(* CODESYS project Elevator0428_RECOVERED_2025-06-24T23-27-54.project

Project tree, tasks and I/O mapping:
  Device : Elmo Platinum Maestro, Elmo Motion Control, version 1.0.0.2
    application Application
      libraries: Standard, * (System); VisuDialogs, * (System)
      task VISU_TASK (cyclic, interval 100 ms, priority 31) calls VisuElems.Visu_Prg, PLC_PRG
      task MainTask (cyclic, interval t#20ms, priority 1) calls nothing
      function block FB_Elevator [ST]: M_IsDoorOpen, M_Enter, M_IsMoving, M_LightState, M_IsAtFloor, M_DisplayNowFloor, M_DisplayNextFloor, M_Move, M_position, M_StopMoving, M_OpenDoor, M_DisElevatorState, M_DisplayDoorState, M_FloorBtnClick, M_CloseDoor
      function block FB_FreightEle [ST]: M_Apperance
      visualisation OutsideEle
      visualisation Elavator
      data type st_Elevator
      interface ITF_Counting: M_Enter
      visualisation FreightElavator
      visualisation Visualization
      interface ITF_Action: M_IsAtFloor, M_Move, M_FloorBtnClick, M_IsDoorOpen, M_position, M_StopMoving, M_IsMoving, M_OpenDoor, M_CloseDoor
      function block FB_PassenEle [ST]
      program PLC_PRG [ST]
      function block FB_Floor [ST]: M_UpBtn, M_CallEleUp, M_CallEleDown, M_Exit, M_DownBtn, M_DeterDirection
      interface ITF_Display: M_DisplayNowFloor, M_LightState, M_DisplayNextFloor, M_DisplayDoorState, M_DisElevatorState
    Maestro : Maestro, Elmo, version 1.0.0.2
  text list GlobalTextList
*)

// Device/Application/st_Elevator
TYPE st_Elevator :
STRUCT
	xKey  : ARRAY [1..5] OF BOOL;
	iFloor: BOOL;
	xEnter : BOOL;
	xExit : BOOL;
	EleState : STRING;
	ODoor :  BOOL;
	CDoor :  BOOL;
	iWay :  STRING;
	iNextFloor : STRING;
	iNowFloor : STRING;
	//ix_Start : BOOL;
END_STRUCT
END_TYPE

// Device/Application/PLC_PRG
PROGRAM PLC_PRG
VAR
	CallELeFloor:INT;
	
	
	fbElevator : ARRAY [1..uiObject] OF FB_Elevator;
	
	fbFreight : FB_FreightEle;
	fbFloors: ARRAY [0..5] OF FB_Floor;
	fbFloorPtrs : ARRAY [0..5] OF POINTER TO FB_Floor;
	
	passoutsideCount: INT:= 5;
	passengerCount : INT := 0;
	
	xKey : ARRAY[1..uiObject] OF BOOL;
	iCnt  : INT;
	bInit : BOOL := FALSE;
	
	curEle : REFERENCE TO FB_Elevator;
	curFloor : INT;
	tmp : INT;
	i: INT;
	j: INT;
	
	CalledElevator : INT;
END_VAR


VAR CONSTANT
	uiObject : INT := 4;
	FloorDistance: INT :=313;
END_VAR

//Ele position and set the positon
IF NOT bInit THEN
	bInit := TRUE;
	
	fbElevator[4] := fbFreight;
	fbElevator[4].minFloor := 0; // Don't know why freight elevator constructor not working
	fbElevator[4].maxCapacity := 5;
	
	
	fbElevator[1].iPos :=945;
	fbElevator[2].iPos :=1258;
	fbElevator[3].iPos :=1258;
	fbElevator[4].iPos :=1258;
	
	fbFloors[0].iPoss := 1571;
	fbFloors[1].iPoss := 1258;
	fbFloors[2].iPoss := 945;
	fbFloors[3].iPoss := 632;
	fbFloors[4].iPoss := 319;
	fbFloors[5].iPoss := 3;
	
	fbFloors[0].FloorNumber := 0;
	fbFloors[1].FloorNumber := 1;
	fbFloors[2].FloorNumber := 2;
	fbFloors[3].FloorNumber := 3;
	fbFloors[4].FloorNumber := 4;
	fbFloors[5].FloorNumber := 5;
	
	FOR i := 0 TO 5 BY 1 DO
		fbFloorPtrs[i]:= ADR(fbFloors[i]);   //pointer to fbFloors (used in fb_elevator)
	END_FOR
	
	FOR i := 1 TO 4 BY 1 DO
		fbElevator[i].FloorNow := fbElevator[i].M_IsAtFloor(fbFloorPtrs);
	END_FOR
	
	FOR i := 1 TO 4 BY 1 DO
		FOR j := 0 TO 5 BY 1 DO
			fbElevator[i].Floorptr[j]:=ADR(fbFloors[j]);  //pointer to fbFloors (store floor info in elevator)
		END_FOR
	END_FOR
		
		
	FOR i := 0 TO 5 BY 1 DO
		FOR j := 1 TO 4 BY 1 DO
			fbFloors[i].fbElevatorPtrs[j]:=ADR(fbElevator[j]);  //pointer to fbelevator (record ele info in Floors )
			fbFloors[i].shouldStop[j] := FALSE;
		END_FOR
	END_FOR	
END_IF

//check ele state: move/ not yet
FOR iCnt := 1 TO uiObject BY 1 DO
	curEle REF= fbElevator[iCnt];  //we are going to change the parameter in curEle some where else, so if not using ref, curEle only will be a clone object (will not update the change)
	IF curEle.M_IsMoving() THEN //moving
		tmp := curEle.M_IsAtFloor(fbFloorPtrs);
		IF  (tmp <> -1) AND tmp = curEle.TargetFloor THEN  //reach the TargetFloor (going to stop)
			fbElevator[iCnt].M_StopMoving();
		ELSE
			IF NOT fbElevator[iCnt].M_IsDoorOpen() THEN //start moving
				curEle.M_Move(fbFloors);
				fbElevator[iCnt].Light := fbElevator[iCnt].M_LightState();
				fbElevator[iCnt].iPos:= curEle.M_position(fbElevator[iCnt].iPos);
			END_IF
		END_IF
		
	ELSE // pending
		curEle.iWaitingCounter := curEle.iWaitingCounter + 1;
		IF NOT curEle.M_IsDoorOpen() OR curEle.iWaitingCounter > curEle.iMaxWaitingTime THEN
			curEle.iWaitingCounter := 0;
			curEle.M_CloseDoor();
			IF NOT (curEle.TargetFloor = -1) THEN  //has target then move
				curEle.M_Move(fbFloors);
				fbElevator[iCnt].Light := fbElevator[iCnt].M_LightState();
				fbElevator[iCnt].iPos:= curEle.M_position(fbElevator[iCnt].iPos);
			END_IF
		END_IF
	END_IF
	
//display part
	fbElevator[iCnt].M_DisplayNowFloor();
	fbElevator[iCnt].M_DisplayNextFloor();
	fbElevator[iCnt].M_DisplayDoorState();
	fbElevator[iCnt].M_DisElevatorState();

	
END_FOR

//see wether elevator has change target floor
(*FOR i := 0 TO 5 BY 1 DO
	IF fbFloors[i].M_UpBtn() OR  fbFloors[i].M_DownBtn() THEN
		CalledElevator := fbFloors[i].M_CallEleUp();
		IF NOT (CalledElevator = -1) THEN
			fbElevator[CalledElevator].M_Move(fbFloors);
		END_IF
	END_IF
END_FOR		*)

END_PROGRAM

// Device/Application/FB_Elevator
FUNCTION_BLOCK FB_Elevator IMPLEMENTS ITF_Action,ITF_Display,ITF_Counting
VAR_INPUT
	ix_Start  : BOOL;
	xKey  : ARRAY [0..5] OF BOOL;
	
	Floorptr: ARRAY[0..5] OF POINTER TO FB_Floor ;
	ODoor : BOOL;
	CDoor : BOOL;
	Enter : BOOL;
	iPos : INT;
	iPoss : INT;
	iWaitingCounter : INT;
	passoutsideCount: INT:= 5;
	passengerCount : INT := 0;
	iMove: INT:=0;
	FloorNow  : INT :=1;
	EleState : STRING;
	Light: BOOL := FALSE; 
	
	TargetFloor  :INT:= -1;
	maxFloor : INT := 5;
	minFloor : INT := 0;
	
	direction : INT := 0;
	maxCapacity : INT := 3;
	
END_VAR
VAR_OUTPUT
	
END_VAR
VAR
	//StrDir:STRING;
	DoMove: BOOL :=FALSE;
	stFloorNow  : STRING;
	stTargetFloor  :STRING :='';
	
	
	doorstate : BOOL := TRUE;  
	DoorDisplay : STRING;
	
	
		turnlight:BOOL;
	
	
	
	
    
	
	
	Speed: INT := 1;
	
	iKeyClicked : INT;
	
	currentFloor: BOOL;
	xEnter : BOOL;
	
	//ODoor :  BOOL;
	//CDoor :  BOOL;
	iWay :  STRING;
	iNextFloor : STRING;
	iNowFloor : STRING;
	
	os_Status : STRING;
	
	xDoorFullyOpen : BOOL;
	fbAutoCloseTimer : TON; 
	tDoorOpenDwellTime : TIME := T#10S;
	bAutoCloseTriggered : BOOL;
	
	bIsMoving : BOOL := FALSE;
	
	
	
	
	iMaxWaitingTime : INT := 50;

END_VAR
VAR CONSTANT
END_VAR

fbAutoCloseTimer.IN := xDoorFullyOpen;
fbAutoCloseTimer.PT := tDoorOpenDwellTime;
fbAutoCloseTimer ();

IF fbAutoCloseTimer.Q AND (DoorState = FALSE) AND NOT bAutoCloseTriggered THEN
	THIS^.M_CloseDoor(); 
	bAutoCloseTriggered := TRUE;
END_IF

maxFloor := 5;
minFloor := 1; // default For passenger Elevator

METHOD M_IsDoorOpen : BOOL
VAR_INPUT
END_VAR
M_IsDoorOpen := doorstate;
END_METHOD

METHOD M_Enter: BOOL
VAR_INPUT
	
END_VAR

VAR
	i:INT;
END_VAR
IF NOT (M_IsAtFloor(Floorptr) = -1) THEN
	IF passengerCount < maxCapacity AND NOT (Floorptr[FloorNow]^.passoutsideCount=0) AND M_IsDoorOpen() THEN
		Floorptr[FloorNow]^.passoutsideCount:=Floorptr[FloorNow]^.passoutsideCount -1 ;
		passengerCount := passengerCount +1;
		M_Enter := TRUE; 
		RETURN;
	END_IF
END_IF

	M_Enter := FALSE;
END_METHOD

METHOD M_IsMoving : BOOL
VAR_INPUT
END_VAR
M_IsMoving := bIsMoving;
END_METHOD

METHOD M_LightState : BOOL
VAR_INPUT
	
END_VAR
IF turnlight THEN
	M_LightState := TRUE;
ELSE
	M_LightState:= FALSE;
END_IF
END_METHOD

METHOD M_IsAtFloor : INT
VAR_INPUT
	fbFloorsPtr : ARRAY[0..5] OF POINTER TO FB_Floor;
END_VAR
VAR
	i : INT;
END_VAR
FOR i := 1 TO 5 BY 1 DO
	IF( ABS(iPos - fbFloorsPtr[i]^.iPoss) < 5) THEN  
		M_IsAtFloor := i;
		FloorNow := M_IsAtFloor;
		RETURN;
	END_IF
END_FOR
M_IsAtFloor := -1; // -1 represents, no floor
END_METHOD

METHOD M_DisplayNowFloor : STRING
VAR_INPUT
END_VAR
IF FloorNow > 0 AND FloorNow < 6 THEN
	M_DisplayNowFloor :=INT_TO_STRING(FloorNow);
	stFloorNow := M_DisplayNowFloor;
ELSIF FloorNow = 0 THEN
	M_DisplayNowFloor :='B1';
	stFloorNow := M_DisplayNowFloor;
ELSE 
	M_DisplayNowFloor := '';
	stFloorNow := M_DisplayNowFloor;
END_IF
END_METHOD

METHOD M_DisplayNextFloor : STRING
VAR_INPUT
END_VAR

VAR
	LastTargetFloor: INT:=6; //initial set as the max floor
	i:INT;
END_VAR
IF TargetFloor < LastTargetFloor THEN
	IF TargetFloor > 0 AND TargetFloor < 6 THEN
		M_DisplayNextFloor :=INT_TO_STRING(TargetFloor);
		stTargetFloor := M_DisplayNextFloor; //
	ELSIF TargetFloor = 0 THEN
		M_DisplayNextFloor :='B1';
		stTargetFloor := M_DisplayNextFloor;
	ELSE 
		M_DisplayNextFloor := '';
		stTargetFloor := M_DisplayNextFloor;
	END_IF
	LastTargetFloor:=TargetFloor;
END_IF
	RETURN;
END_METHOD

METHOD M_Move : INT
VAR_INPUT
	fbFloors : ARRAY[0..5] OF FB_Floor;
END_VAR
VAR
	target_pos : INT;
	i : INT;
	hasNextFloor : BOOL;
	lastdirect : INT;
END_VAR
bIsMoving := TRUE;


// Change direction
IF NOT (TargetFloor = -1) THEN
	//Light := TRUE;
	target_pos := fbFloors[TargetFloor].iPoss;   
	IF target_pos < iPos THEN
		direction := -1;  //DOWN
		turnlight:= TRUE;
	ELSIF target_pos > iPos THEN
		direction := 1; //UP
		turnlight:= TRUE;
	ELSE
		//direction := 0;
		turnlight:= FALSE;
	END_IF
	lastdirect:= direction;  // lastdirect for 
//not END_IF yet

	IF NOT ( ABS(iPos - target_pos) < 5) THEN
		iMove := iMove + THIS^.direction * speed;
	ELSE
		//reach target, reset
		turnlight := FALSE;
		FloorNow := M_IsAtFloor(FloorPtr);
		xKey[TargetFloor] := FALSE;
		TargetFloor := -1;
		
		
		// check whether there is next target floor
		hasNextFloor := FALSE;  
		FOR i := 0 TO 5 BY 1 DO
			IF xKey[i] THEN  //if there is still any being pressed, deal with the next target floor
				hasNextFloor := TRUE;
				EXIT; 
			END_IF
		END_FOR
		
	// Enter the next targer floor 
		
		IF hasNextFloor THEN
			IF direction = 1 THEN   //find up way first
				FOR i := FloorNow + 1 TO maxFloor BY 1 DO   
					IF xKey[i] THEN
						TargetFloor := i;
						EXIT;
					END_IF
				END_FOR
				IF TargetFloor = -1 THEN
					FOR i := FloorNow - 1 TO minFloor BY -1 DO
						IF xKey[i] THEN
							TargetFloor := i;
							EXIT;
						END_IF
					END_FOR
				END_IF
			ELSIF direction = -1 THEN  //or find down way 
				FOR i := FloorNow - 1 TO minFloor BY -1 DO
					IF xKey[i] THEN
						TargetFloor := i;
						EXIT;
					END_IF
				END_FOR
				IF TargetFloor = -1 THEN
					FOR i := FloorNow + 1 TO maxFloor BY 1 DO
						IF xKey[i] THEN
							TargetFloor := i;
							EXIT;
						END_IF
					END_FOR
				END_IF
			ELSE
				// should not happen
			END_IF
		END_IF
		
	//NO FloorBtn is on, looking for upBtn at any floor
		IF TargetFloor = -1 THEN 
			
				FOR i := 1 TO 5 BY 1 DO 
				 // check the floor , i represent floor dis
					IF FloorNow + i <= maxFloor THEN
						// M_UpBtn and M_DownBtn methods will change the button state
						////IF Floorptr[FloorNow + i]^.M_UpBtn() AND NOT Floorptr[FloorNow + i]^.UpEleGet THEN
						IF Floorptr[FloorNow + i]^.xUp AND NOT Floorptr[FloorNow + i]^.UpSolved THEN
							TargetFloor := FloorNow + i;
							Floorptr[FloorNow + i]^.UpSolved := TRUE;
							//Floorptr[FloorNow + i]^.xUp := TRUE;
							EXIT;
						////ELSIF  Floorptr[FloorNow + i]^.M_DownBtn() AND NOT Floorptr[FloorNow + i]^.DownEleGet THEN
						ELSIF  Floorptr[FloorNow + i]^.xDown AND NOT Floorptr[FloorNow + i]^.DownSolved THEN
							TargetFloor := FloorNow + i;
							Floorptr[FloorNow + i]^.DownSolved:= TRUE;
							//Floorptr[FloorNow + i]^.xDown := TRUE;
							EXIT;
						END_IF
					END_IF
					
					
					IF FloorNow - i >= minFloor THEN
						// M_UpBtn and M_DownBtn methods will change the button state			
						////IF Floorptr[FloorNow - i]^.M_UpBtn() AND NOT Floorptr[FloorNow - i]^.UpEleGet THEN
						IF Floorptr[FloorNow - i]^.xUp AND NOT Floorptr[FloorNow - i]^.UpSolved THEN
							TargetFloor := FloorNow - i;
							Floorptr[FloorNow - i]^.UpSolved:= TRUE;
							//Floorptr[FloorNow - i]^.xUp := TRUE;
							EXIT;
						////ELSIF  Floorptr[FloorNow - i]^.M_DownBtn() AND NOT Floorptr[FloorNow - i]^.DownEleGet THEN
						ELSIF  Floorptr[FloorNow - i]^.xDown AND NOT Floorptr[FloorNow - i]^.DownSolved THEN
							TargetFloor := FloorNow - i;
							Floorptr[FloorNow - i]^.DownSolved:= TRUE;
							//Floorptr[FloorNow - i]^.xDown := TRUE;
							EXIT;
						END_IF
					END_IF
								
				END_FOR
		END_IF
			
					
				
		//Ele just arrived, stop moving and open door
		M_StopMoving();
		M_OpenDoor();
	END_IF
END_IF //end_if is here
M_Move := iMove;
END_METHOD

METHOD M_position : INT
VAR_INPUT
	In_iPos: INT; 
END_VAR
In_iPos := In_iPos + direction * speed;
M_position := In_iPos;
END_METHOD

METHOD M_StopMoving
VAR_INPUT
END_VAR
iWaitingCounter := 0;
bIsMoving := FALSE;
Light := FALSE;
END_METHOD

METHOD M_OpenDoor : BOOL
VAR_INPUT
	
END_VAR
IF turnlight THEN
	doorstate:= FALSE;
ELSE
	doorstate:= TRUE;
END_IF

M_OpenDoor :=doorstate;
END_METHOD

METHOD M_DisElevatorState : STRING
VAR_INPUT
END_VAR

VAR_IN_OUT
END_VAR

VAR
	StrDir : STRING;
END_VAR
IF turnlight THEN
	IF THIS^.direction = -1 THEN
		StrDir := 'Going Up';
	ELSIF THIS^.direction =1 THEN
		StrDir := 'Going Down';
	END_IF
ELSE
	StrDir := 'Pending';
END_IF

THIS^.EleState := StrDir;
M_DisElevatorState := StrDir;
END_METHOD

METHOD M_DisplayDoorState : STRING
VAR_INPUT
END_VAR
IF doorstate THEN
	DoorDisplay := 'Open';
ELSE
	DoorDisplay := 'Close';
END_IF;
M_DisplayDoorState := DoorDisplay;

(*IF ODoor THEN
	DoorDisplay:='Open';
	doorstate:= TRUE;
ELSIF CDoor THEN
	DoorDisplay:='Close';
	doorstate:= FALSE;
END_IF*)
END_METHOD

METHOD M_FloorBtnClick : BOOL
VAR_INPUT
	xNumber  : INT;
END_VAR

VAR
	fbFloors : ARRAY[0..5] OF FB_Floor;
	btnPos : INT;
	targetPos : INT;
	curPos : INT;
END_VAR
fbFloors[0].iPoss := 1571;
fbFloors[1].iPoss := 1258;
fbFloors[2].iPoss := 945;
fbFloors[3].iPoss := 632;
fbFloors[4].iPoss := 319;
fbFloors[5].iPoss := 3;

IF xNumber < 0 OR xNumber > 5 THEN
	M_FloorBtnClick := FALSE;
	RETURN;
END_IF

//no targer floor and not moving yet
IF (NOT M_IsMoving()) AND TargetFloor = -1 THEN
	TargetFloor :=xNumber;
	xKey[xNumber]:=TRUE;
	bIsMoving := TRUE;

//already have TargetFloor
ELSIF NOT (TargetFloor = -1) THEN
	btnPos := fbFloors[xNumber].iPoss;
	targetPos := fBFloors[TargetFloor].iPoss;
	curPos := iPos;
	IF NOT xKey[xNumber] THEN
		xKey[xNumber] := TRUE;
		IF TargetFloor = xNumber THEN 
			// do nothing
		ELSIF curPos <= btnPos AND btnPos <= targetPos THEN  //ex: now at 2nd btnPos= 4, targetPos= 5
			TargetFloor := xNumber;  // TargetFloor update to btnPos= 4
		ELSIF curPos >= btnPos AND btnPos >= targetPos THEN  // same as above but downstairs
			TargetFloor := xNumber;
		END_IF
	ELSE 
		// try to cancel btn, not supported now
	END_IF
END_IF
END_METHOD

METHOD M_CloseDoor : BOOL
VAR_INPUT
END_VAR
doorstate := FALSE;
M_CloseDoor := doorstate;
END_METHOD

END_FUNCTION_BLOCK

// Device/Application/ITF_Action
INTERFACE ITF_Action

METHOD M_IsAtFloor : INT
VAR_INPUT
	fbFloorsPtr : ARRAY[0..5] OF POINTER TO FB_Floor;
END_VAR
END_METHOD

METHOD M_Move : INT
VAR_INPUT
	fbFloors : ARRAY[0..5] OF FB_Floor;
END_VAR
END_METHOD

METHOD M_FloorBtnClick : BOOL
VAR_INPUT
	xNumber  : INT;
END_VAR
END_METHOD

METHOD M_IsDoorOpen : BOOL
VAR_INPUT
END_VAR
END_METHOD

METHOD M_position : INT
VAR_INPUT
	In_iPos: INT; 
END_VAR
END_METHOD

METHOD M_StopMoving
VAR_INPUT
END_VAR
END_METHOD

METHOD M_IsMoving : BOOL
VAR_INPUT
END_VAR
END_METHOD

METHOD M_OpenDoor : BOOL
VAR_INPUT
END_VAR
END_METHOD

METHOD M_CloseDoor : BOOL
VAR_INPUT
END_VAR
END_METHOD

END_INTERFACE

// Device/Application/FB_Floor
FUNCTION_BLOCK FB_Floor 
VAR_INPUT
	
	FloorNumber : INT; // This indicates which floor current FB_Floor object is.

	iPoss : INT;
	passOutsideCount : INT:=5;
	
	fbElevatorPtrs : ARRAY[1..4] OF POINTER TO FB_Elevator;
	
	shouldStop : ARRAY[1..4] OF BOOL;
	
	UpEleGet : BOOL:= FALSE;
	DownEleGet : BOOL:= FALSE;
	
	UpSolved : BOOL := FALSE;
	DownSolved : BOOL := FALSE;
	
	xUp : BOOL;
	xDown : BOOL;
	
END_VAR
VAR
	
	
	
	
	xExit : BOOL;
	
	EleState : STRING;
		
END_VAR

METHOD M_UpBtn : BOOL
VAR_INPUT
END_VAR
VAR
	i:INT;
	PendingElevator: ARRAY [1..4] OF INT;
	FloorDis: ARRAY [1..4] OF INT;
	
	shortest:INT;
	EleWantedNumber : INT := -1;
END_VAR
IF xUp = TRUE OR (NOT xUp AND UpSolved) THEN
	RETURN;
END_IF

UpSolved := FALSE;
xUp:= TRUE;
//UpEleGet:= FALSE;

FOR i := 1 TO 4 BY 1 DO
// elevator moving or not
	IF  NOT fbElevatorPtrs[i]^.turnlight THEN
		PendingElevator[i]:= 1; //pending ELe
	ELSE
		PendingElevator[i]:= 0; //moving ELe
	END_IF
END_FOR

shortest := 20000;
EleWantedNumber := -1; //no elevator is assigned to come
FOR i := 1 TO 4 BY 1 DO
//Pending ELe, then pick a nearer one
	IF PendingElevator[i] = 1 THEN
		FloorDis[i]:=ABS(fbElevatorPtrs[i]^.iPos - iPoss);
		
		IF FloorDis[i] < shortest THEN
			shortest := FloorDis[i];
			EleWantedNumber := i;
			UpSolved := TRUE;
			xUp := FALSE;
		END_IF
	
	END_IF
END_FOR

IF EleWantedNumber = -1 THEN
	FOR i := 1 TO 4 BY 1 DO
		//moving ELe, comfirm Ele is two floor away
		IF PendingElevator[i] = 0 AND fbElevatorPtrs[i]^.direction =1 THEN
			IF fbElevatorPtrs[i]^.TargetFloor >= FloorNumber THEN		
				IF ABS(fbElevatorPtrs[i]^.iPos - iPoss >= 626) THEN
					EleWantedNumber:= i;  // no.i elevator needs to come
					UpSolved := TRUE;
					xUp := FALSE;
					EXIT;
				END_IF
			END_IF
		END_IF
	END_FOR
END_IF

IF (EleWantedNumber <>-1) THEN
	fbElevatorPtrs[EleWantedNumber]^.TargetFloor := FloorNumber;
END_IF

//IF (fbElevatorPtrs[EleWantedNumber]^.TargetFloor = FloorNumber) AND (fbElevatorPtrs[EleWantedNumber]^.M_IsDoorOpen) THEN
    //bUpRequested := FALSE;
//END_IF
//M_UpBtn:=xUp;
END_METHOD

METHOD M_CallEleUp :INT
VAR_INPUT
END_VAR
VAR
	i:INT;
	PendingElevator: ARRAY [1..4] OF INT;
	FloorDis: ARRAY [1..4] OF INT;
	
	shortest:INT;
	EleWantedNumber : INT := -1;
	
END_VAR
FOR i := 1 TO 4 BY 1 DO
// elevator moving or not
	IF  fbElevatorPtrs[i]^.turnlight THEN
		PendingElevator[i]:= 1; //pending ELe
	ELSE
		PendingElevator[i]:= 0; //moving ELe
	END_IF
END_FOR

shortest := 2000;
EleWantedNumber := -1; //no elevator is assigned to come
FOR i := 1 TO 4 BY 1 DO
//Pending ELe, then pick a nearer one
	IF PendingElevator[i] = 1 THEN
		FloorDis[i]:=ABS(fbElevatorPtrs[i]^.iPos - iPoss);
		
		IF FloorDis[i] < shortest THEN
			shortest := FloorDis[i];
			EleWantedNumber := i;
		END_IF
	
	END_IF
END_FOR

IF EleWantedNumber = -1 THEN
	FOR i := 1 TO 4 BY 1 DO
		//moving ELe, comfirm Ele is two floor away
		IF PendingElevator[i] = 0 AND fbElevatorPtrs[i]^.direction =1 THEN
			IF ABS(fbElevatorPtrs[i]^.iPos - iPoss >= 621) THEN
				EleWantedNumber:= i;  // no.i elevator needs to come
				EXIT;
			END_IF
		END_IF
	END_FOR
END_IF

M_CallEleUp:= EleWantedNumber;

//when reaching targetfloor, Btn light went out
END_METHOD

METHOD M_CallEleDown : INT
VAR_INPUT
END_VAR
VAR
	i:INT;
	PendingElevator: ARRAY [1..4] OF INT;
	FloorDis: ARRAY [1..4] OF INT;
	
	shortest:INT;
	EleWantedNumber : INT := -1;
	
END_VAR
FOR i := 1 TO 4 BY 1 DO
// elevator moving or not
	IF  fbElevatorPtrs[i]^.turnlight THEN
		PendingElevator[i]:= 1; //pending ELe
	ELSE
		PendingElevator[i]:= 0; //moving ELe
	END_IF
END_FOR

shortest := 2000;
EleWantedNumber := -1; //no elevator is assigned to come
FOR i := 1 TO 4 BY 1 DO
//Pending ELe, then pick a nearer one
	IF PendingElevator[i] = 1 THEN
		FloorDis[i]:=ABS(fbElevatorPtrs[i]^.iPos - iPoss);
		
		IF FloorDis[i] < shortest THEN
			shortest := FloorDis[i];
			EleWantedNumber := i;
			DownSolved:=TRUE;
		END_IF
	
	END_IF
END_FOR

IF EleWantedNumber = -1 THEN
	FOR i := 1 TO 4 BY 1 DO
		//moving ELe, comfirm Ele is two floor away
		IF PendingElevator[i] = 0 AND fbElevatorPtrs[i]^.direction =-1 THEN
			IF ABS(fbElevatorPtrs[i]^.iPos - iPoss >= 626) THEN
				EleWantedNumber:= i;  // no.i elevator needs to come
				DownSolved:=TRUE;
			EXIT;
			END_IF
		END_IF
	END_FOR
END_IF

M_CallEleDown:= EleWantedNumber;

//when reaching targetfloor, Btn light went out
END_METHOD

METHOD M_Exit : BOOL
VAR_INPUT
	
END_VAR
VAR
	i: INT;
END_VAR
FOR i := 1 TO 4 BY 1 DO   
	IF ( ABS(iPoss - fbElevatorPtrs[i]^.iPos) < 5) AND fbElevatorPtrs[i]^.M_IsDoorOpen() THEN
		IF fbElevatorPtrs[i]^.passengerCount > 0 AND fbElevatorPtrs[i]^.passengerCount <8 THEN
			fbElevatorPtrs[i]^.passengerCount:= fbElevatorPtrs[i]^.passengerCount-1;
			passoutsideCount:=passoutsideCount +1;
		END_IF
	END_IF
END_FOR	
(*IF passoutsideCount > 0 THEN
		FloorRef0.passoutsideCount:=FloorRef0.passoutsideCount-1;
		passengerCount := passengerCount +1;
		M_Enter := TRUE; 
	   END_IF

CASE FloorNow OF
	0: 
	
	1: IF passengerCount < maxCapacity AND NOT (FloorRef1.passoutsideCount=0) THEN
		FloorRef1.passoutsideCount:=FloorRef1.passoutsideCount-1;
		passengerCount := passengerCount +1;
		M_Enter := TRUE; 
		RETURN;
	   END_IF
	   
	2: IF passengerCount < maxCapacity AND NOT (FloorRef2.passoutsideCount=0) THEN
		FloorRef2.passoutsideCount:=FloorRef2.passoutsideCount-1;
		passengerCount := passengerCount +1;
		M_Enter := TRUE; 
		RETURN;
	   END_IF
	 
	3: IF passengerCount < maxCapacity AND NOT (FloorRef3.passoutsideCount=0) THEN
		FloorRef3.passoutsideCount:=FloorRef3.passoutsideCount-1;
		passengerCount := passengerCount +1;
		M_Enter := TRUE; 
		RETURN;
	   END_IF
	
	4: IF passengerCount < maxCapacity AND NOT (FloorRef4.passoutsideCount=0) THEN
		FloorRef4.passoutsideCount:=FloorRef4.passoutsideCount-1;
		passengerCount := passengerCount +1;
		M_Enter := TRUE; 
		RETURN;
	   END_IF
	5: IF passengerCount < maxCapacity AND NOT (FloorRef5.passoutsideCount=0) THEN
		FloorRef5.passoutsideCount:=FloorRef5.passoutsideCount-1;
		passengerCount := passengerCount +1;
		M_Enter := TRUE; 
		RETURN;
	   END_IF
	END_CASE

	M_Enter := FALSE; *)
END_METHOD

METHOD M_DownBtn : BOOL
VAR_INPUT
END_VAR
VAR
	i:INT;
	PendingElevator: ARRAY [1..4] OF INT;
	FloorDis: ARRAY [1..4] OF INT;
	
	shortest:INT;
	EleWantedNumber : INT := -1;
	
END_VAR
IF xDown = TRUE OR (NOT xDown AND DownSolved) THEN
	RETURN;
END_IF

xDown:= TRUE;
DownSolved:=FALSE;

FOR i := 1 TO 4 BY 1 DO
// elevator moving or not
	IF NOT fbElevatorPtrs[i]^.turnlight THEN
		PendingElevator[i]:= 1; //pending ELe
	ELSE
		PendingElevator[i]:= 0; //moving ELe
	END_IF
END_FOR

shortest := 20000;
EleWantedNumber := -1; //no elevator is assigned to come
FOR i := 1 TO 4 BY 1 DO
//Pending ELe, then pick a nearer one
	IF PendingElevator[i] = 1 THEN
		FloorDis[i]:=ABS(fbElevatorPtrs[i]^.iPos - iPoss);
		
		IF FloorDis[i] < shortest THEN
			shortest := FloorDis[i];
			EleWantedNumber := i;
			DownSolved := TRUE;
			xDown:= FALSE;
		END_IF
	
	END_IF
END_FOR

IF EleWantedNumber = -1 THEN
	FOR i := 1 TO 4 BY 1 DO
		//moving ELe, comfirm Ele is two floor away
		IF PendingElevator[i] = 0 AND fbElevatorPtrs[i]^.direction =-1 THEN
			IF fbElevatorPtrs[i]^.TargetFloor <= FloorNumber THEN
				IF fbElevatorPtrs[i]^.iPos - iPoss >= 626 THEN
					EleWantedNumber:= i;  // no.i elevator needs to come
					DownSolved := TRUE;
					xDown:= FALSE;
					EXIT;
				END_IF
			END_IF
		END_IF
	END_FOR
END_IF

IF NOT (EleWantedNumber= -1 )THEN
	fbElevatorPtrs[EleWantedNumber]^.TargetFloor := FloorNumber;
END_IF


//M_CallEleDown:= EleWantedNumber;

//when reaching targetfloor, Btn light went out

	
//M_DownBtn:=xDown;
END_METHOD

METHOD M_DeterDirection
VAR_INPUT
END_VAR
(*IF xUp  THEN
        direction := 1;
		Light := TRUE;
		
ELSIF xDown THEN
        direction := -1;
		Light := TRUE;
ELSE
        direction := 0;
		Light := FALSE;
END_IF;   *)
END_METHOD

END_FUNCTION_BLOCK

// Device/Application/ITF_Display
INTERFACE ITF_Display

METHOD M_DisplayNowFloor : STRING
VAR_INPUT
END_VAR
END_METHOD

METHOD M_LightState : BOOL
VAR_INPUT
	
END_VAR
END_METHOD

METHOD M_DisplayNextFloor : STRING
VAR_INPUT
END_VAR
END_METHOD

METHOD M_DisplayDoorState : STRING
VAR_INPUT
END_VAR
END_METHOD

METHOD M_DisElevatorState : STRING
VAR_INPUT
END_VAR

VAR_IN_OUT
END_VAR
END_METHOD

END_INTERFACE

// Device/Application/ITF_Counting
INTERFACE ITF_Counting

METHOD M_Enter : BOOL
VAR_INPUT
END_VAR
END_METHOD

END_INTERFACE

// Device/Application/FB_FreightEle
FUNCTION_BLOCK FB_FreightEle EXTENDS FB_Elevator
VAR_INPUT
	
END_VAR
VAR_OUTPUT
END_VAR
VAR
END_VAR

//SUPER^();
maxFloor := 5;
minFloor := 0;
maxCapacity := 5;

METHOD M_Apperance
VAR_INPUT
END_VAR
END_METHOD

END_FUNCTION_BLOCK

// Device/Application/FB_PassenEle
FUNCTION_BLOCK FB_PassenEle EXTENDS FB_Elevator 
VAR_INPUT
END_VAR
VAR_OUTPUT
END_VAR
VAR
	
END_VAR

SUPER^();
maxFloor := 5;
minFloor := 1; // default For passenger Elevator

END_FUNCTION_BLOCK

// Device/Application/OutsideEle
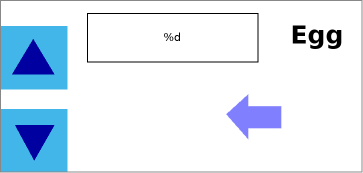
VISUALIZATION OutsideEle  // 363x173
VAR_IN_OUT
	fbFloorsVisu  : fb_Floor;
END_VAR
    RoundedRectangle (1,26 66x63)
        tap fbFloorsVisu.xUp
        OnMouseClick: execute { fbFloorsVisu.M_UpBtn(); }
    Polygon (33,39) (12,74) (54,74)
    RoundedRectangle (1,109 66x63)
        tap fbFloorsVisu.xDown
        OnMouseClick: execute { fbFloorsVisu.M_DownBtn(); }
    Polygon (15,125) (34,160) (54,125)
    Rectangle (87,13 171x49), "%d", text variable: fbFloorsVisu.passoutsideCount
    Label (292,13 50x43), "Egg"
    Polygon (226,114) (248,94) (248,106) (281,106) (281,128) (248,128) (248,139), text variable: fbFloorsVisu.xExit
        tap fbFloorsVisu.xExit
        OnMouseClick: execute { fbFloorsVisu.M_Exit(); }
END_VISUALIZATION

// Device/Application/Elavator
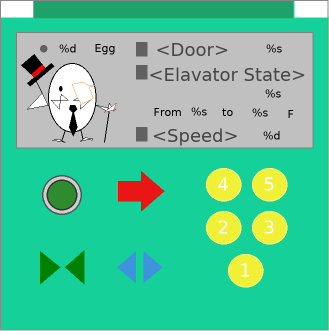
VISUALIZATION Elavator  // 329x331
VAR_IN_OUT
	fbElevatorVisu  : fb_Elevator;
END_VAR
    Polyline (46,537) (47,538)
    RoundedRectangle (0,17 329x313)
    RoundedRectangle (16,32 297x116)
    Ellipse (252,168 35x33), "5"
        tap fbElevatorVisu.xKey[5]
        OnMouseClick: execute { fbElevatorVisu.M_FloorBtnClick(5); }
    Ellipse (252,211 35x33), "3"
        tap fbElevatorVisu.xKey[3]
        OnMouseClick: execute { fbElevatorVisu.M_FloorBtnClick(3); }
    Ellipse (206,168 35x33), "4"
        tap fbElevatorVisu.xKey[4]
        OnMouseClick: execute { fbElevatorVisu.M_FloorBtnClick(4); }
    Ellipse (206,211 35x33), "2"
        tap fbElevatorVisu.xKey[2]
        OnMouseClick: execute { fbElevatorVisu.M_FloorBtnClick(2); }
    Ellipse (228,254 35x33), "1"
        tap fbElevatorVisu.xKey[1]
        OnMouseClick: execute { fbElevatorVisu.M_FloorBtnClick(1); }
    Lamp1 (39,170 46x50), variable: fbElevatorVisu.Light, style: Lamp-Lamp1-Green
    Polygon (141,171) (164,191) (141,211) (141,201) (118,201) (118,181) (141,181)
        tap fbElevatorVisu.xEnter
        OnMouseClick: execute { fbElevatorVisu.M_Enter(); }
    Rectangle (37,39 62x20), "%d", text variable: fbElevatorVisu.passengerCount
    Rectangle (136,42 11x14)
    Label (108,37 169x26), "<Door>"
    Rectangle (237,40 74x18), "%s", text variable: fbElevatorVisu.DoorDisplay
    Rectangle (223,104 74x18), "%s", text variable: fbElevatorVisu.stTargetFloor
    Rectangle (136,65 11x14)
    Label (143,62 169x26), "<Elavator State>"
    Rectangle (236,85 74x18), "%s", text variable: fbElevatorVisu.EleState
    Label (277,106 28x17), "F"
    Label (85,30 40x37), "Egg"
    Ellipse (40,45 7x7)
    Rectangle (33,0 261x19)
    Group (21,54 95x88)
        Ellipse (27,9 48x69)
        Line (41,86) (44,77)
        Line (62,85) (60,76)
        Ellipse (38,32 3x5)
        Ellipse (56,32 3x5)
        Polygon (75,51) (86,57) (88,49) (92,55)
        Polygon (69,46) (59,55) (61,42) (52,46)
        Polygon (30,46) (38,55) (40,40) (47,46)
        Polygon (15,27) (21,39) (6,55) (27,51)
        Polygon (59,87) (65,83) (71,86) (71,84)
        Line (88,55) (83,88)
        Polygon (83,58) (95,49) (92,57) (95,55)
        Polygon (31,86) (39,85) (39,86) (44,88)
        Polygon (9,32) (33,12) (30,9) (24,14) (13,0) (0,11) (13,23) (6,29)
        Polygon (13,24) (24,14) (21,10) (10,20) (13,23)
        Polygon (68,33) (72,44) (60,50) (55,41) (51,30) (62,28) (67,31) (75,31)
        Group (48,51 4x23)
            Polygon (1,0) (6,0) (8,4) (4,8) (0,4)
            Polygon (4,5) (8,22) (4,31) (0,22)
    Rectangle (162,103 74x18), "%s", text variable: fbElevatorVisu.stFloorNow
        OnMouseClick: write the text variable via Default
    Label (214,104 27x17), "to"
    Label (153,104 29x17), "From"
    Rectangle (136,127 11x14)
    Label (111,123 169x26), "<Speed>"
    Rectangle (235,127 74x18), "%d", text variable: fbElevatorVisu.Speed
        OnMouseClick: write the text variable via Default
    Polygon (137,250) (142,250) (162,267) (142,284) (137,284) (137,284) (117,267)
        tap fbElevatorVisu.ODoor
        OnMouseClick: execute { fbElevatorVisu.M_OpenDoor(); }
    Rectangle (136,240 7x50)
    Polygon (84,250) (84,284) (65,267) (60,267) (40,284) (40,251) (60,267) (65,267)
        tap fbElevatorVisu.CDoor
        OnMouseClick: execute { fbElevatorVisu.M_CloseDoor(); }
    Rectangle (61,241 3x50)
END_VISUALIZATION

// Device/Application/FreightElavator
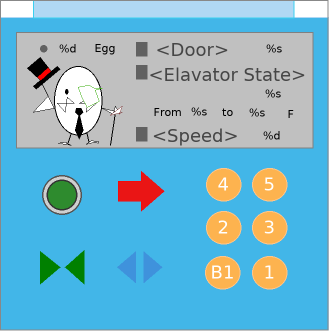
VISUALIZATION FreightElavator  // 329x331
VAR_IN_OUT
	fbFreightVisu  : FB_Elevator;
END_VAR
    Polyline (46,537) (47,538)
    RoundedRectangle (0,17 329x313)
    RoundedRectangle (16,32 297x116)
    Ellipse (252,168 35x33), "5"
        tap fbFreightVisu.xKey[5]
        OnMouseClick: execute { fbFreightVisu.M_FloorBtnClick(5); }
    Ellipse (252,211 35x33), "3"
        tap fbFreightVisu.xKey[3]
        OnMouseClick: execute { fbFreightVisu.M_FloorBtnClick(3); }
    Ellipse (206,168 35x33), "4"
        tap fbFreightVisu.xKey[4]
        OnMouseClick: execute { fbFreightVisu.M_FloorBtnClick(4); }
    Ellipse (206,211 35x33), "2"
        tap fbFreightVisu.xKey[2]
        OnMouseClick: execute { fbFreightVisu.M_FloorBtnClick(2); }
    Ellipse (252,256 35x33), "1"
        tap fbFreightVisu.xKey[1]
        OnMouseClick: execute { fbFreightVisu.M_FloorBtnClick(1); }
    Lamp1 (39,170 46x50), variable: fbFreightVisu.Light, style: Lamp-Lamp1-Green
    Polygon (141,171) (164,191) (141,211) (141,201) (118,201) (118,181) (141,181)
        tap fbFreightVisu.xEnter
        OnMouseClick: execute { fbFreightVisu.M_Enter(); }
    Rectangle (37,39 62x20), "%d", text variable: fbFreightVisu.passengerCount
    Rectangle (136,42 11x14)
    Label (108,37 169x26), "<Door>"
    Rectangle (237,40 74x18), "%s", text variable: fbFreightVisu.DoorDisplay
    Rectangle (220,104 74x18), "%s", text variable: fbFreightVisu.stTargetFloor
    Rectangle (136,65 11x14)
    Label (143,62 169x26), "<Elavator State>"
    Rectangle (236,85 74x18), "%s", text variable: fbFreightVisu.EleState
    Label (277,106 28x17), "F"
    Label (85,30 40x37), "Egg"
    Ellipse (40,45 7x7)
    Rectangle (33,-1 261x19)
    Group (27,57 95x88)
        Ellipse (27,9 48x69)
        Line (41,86) (44,77)
        Line (62,85) (60,76)
        Ellipse (38,32 3x5)
        Ellipse (56,32 3x5)
        Polygon (75,51) (86,57) (88,49) (92,55)
        Polygon (69,46) (59,55) (61,42) (52,46)
        Polygon (30,46) (38,55) (40,40) (47,46)
        Polygon (15,27) (21,39) (6,55) (27,51)
        Polygon (59,87) (65,83) (71,86) (71,84)
        Line (88,55) (83,88)
        Polygon (83,58) (95,49) (92,57) (95,55)
        Polygon (31,86) (39,85) (39,86) (44,88)
        Polygon (9,32) (33,12) (30,9) (24,14) (13,0) (0,11) (13,23) (6,29)
        Polygon (13,24) (24,14) (21,10) (10,20) (13,23)
        Polygon (68,33) (72,44) (60,50) (55,41) (51,30) (62,28) (67,31) (75,31)
        Group (48,51 4x23)
            Polygon (1,0) (6,0) (8,4) (4,8) (0,4)
            Polygon (4,5) (8,22) (4,31) (0,22)
    Rectangle (162,103 74x18), "%s", text variable: fbFreightVisu.stFloorNow
        OnMouseClick: write the text variable via Default
    Label (214,104 27x17), "to"
    Label (153,104 29x17), "From"
    Rectangle (136,127 11x14)
    Label (111,123 169x26), "<Speed>"
    Rectangle (235,127 74x18), "%d", text variable: fbFreightVisu.Speed
        OnMouseClick: write the text variable via Default
    Polygon (137,250) (142,250) (162,267) (142,284) (137,284) (137,284) (117,267)
        tap fbFreightVisu.ODoor
        OnMouseClick: execute { fbFreightVisu.M_OpenDoor(); }
    Rectangle (136,240 7x50)
    Polygon (84,250) (84,284) (65,267) (60,267) (40,284) (40,251) (60,267) (65,267)
        tap fbFreightVisu.CDoor
        OnMouseClick: execute { fbFreightVisu.M_CloseDoor(); }
    Rectangle (61,241 3x50)
    Ellipse (205,256 35x33), "B1"
        tap fbFreightVisu.xKey[0]
        OnMouseClick: execute { fbFreightVisu.M_FloorBtnClick(0); }
END_VISUALIZATION

// Device/Application/Visualization
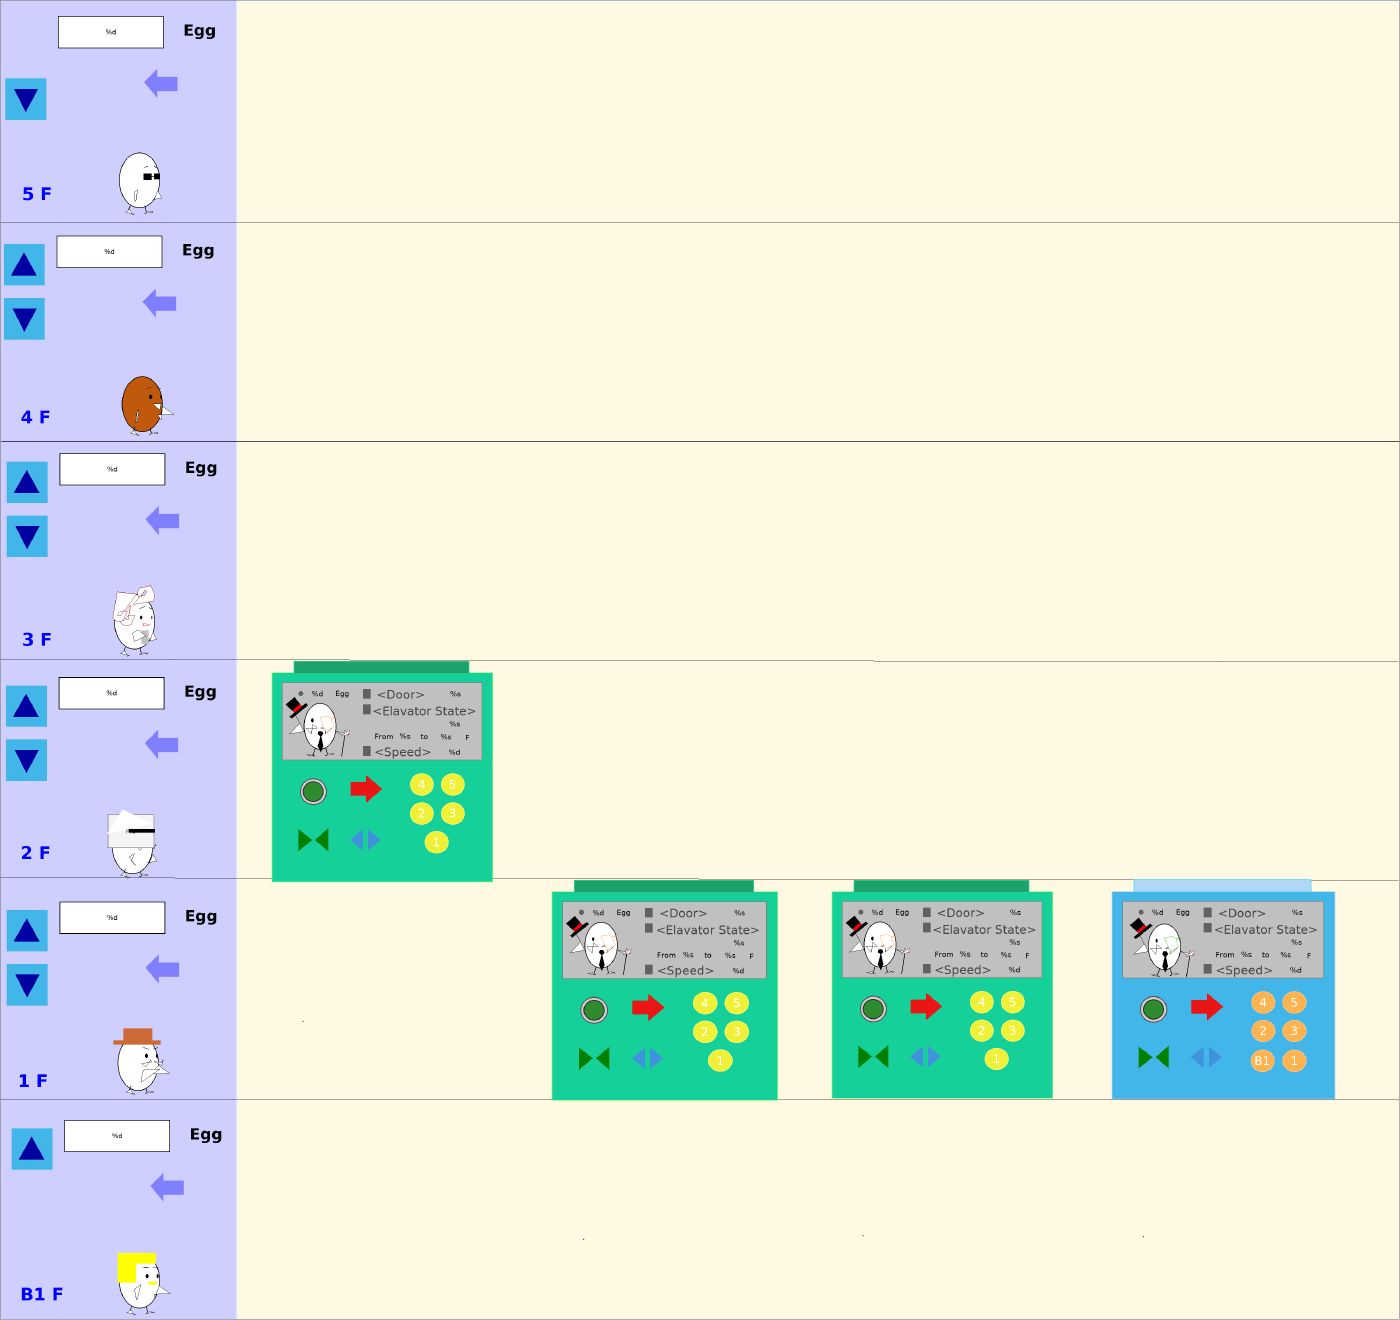
VISUALIZATION Visualization  // 2000x1887
    Rectangle (-4,0 342x1887)
    Rectangle (338,3 1661x1886)
    Line (0,1254) (1997,1258)
    Line (0,942) (1997,946)
    Line (2,631) (2000,631)
    Line (-3,317) (1999,318)
    Line (-2,1571) (1998,1572)
    Frame (788,1258 323x316)
        shows Elavator(fbElevatorVisu := PLC_PRG.fbElevator[2])
        p2738717112: PLC_PRG.fbElevator[2].iMove
    Frame (1188,1258 316x313)
        shows Elavator(fbElevatorVisu := PLC_PRG.fbElevator[3])
        p2738717112: PLC_PRG.fbElevator[3].iMove
    Group (162,1470 80x95)
        Line (48,91) (46,82)
        Polygon (45,93) (51,89) (57,92) (57,90)
        Ellipse (6,10 58x79)
        Polygon (55,63) (57,65) (80,64) (64,53)
        Polygon (44,58) (41,64) (40,77) (66,58)
        Line (22,90) (25,82)
        Polygon (18,91) (24,87) (28,95) (31,94)
        Rectangle (0,17 67x6)
        Rectangle (14,0 41x17)
        Polygon (58,47) (69,53) (71,45) (69,49)
        Polygon (40,50) (46,55) (53,45) (54,48)
        Ellipse (45,36 4x6)
        Ellipse (61,36 2x6)
        Line (50,30) (42,27)
        Line (57,29) (63,27)
    Group (153,1157 71x98)
        Line (49,94) (47,85)
        Polygon (46,96) (52,92) (58,95) (58,93)
        Ellipse (7,13 58x79)
        Polygon (60,77) (58,76) (71,74) (65,64)
        Polygon (39,63) (31,68) (41,80) (34,74)
        Line (23,93) (26,85)
        Polygon (19,94) (25,90) (29,98) (32,97)
        Polygon (59,50) (67,56) (69,50) (70,52)
        Polygon (42,54) (47,58) (54,48) (55,51)
        Ellipse (46,39 4x6)
        Ellipse (62,39 2x6)
        Line (51,33) (44,35)
        Line (58,32) (63,35)
        Pie (1,7 66x48)
        Rectangle (31,28 37x5)
        Polygon (63,20) (22,0) (0,35) (0,35)
    Group (161,837 63x101)
        Ellipse (2,12 58x79)
        Line (41,97) (39,88)
        Polygon (38,99) (44,95) (50,98) (50,96)
        Polygon (52,80) (50,79) (63,77) (57,67)
        Line (15,96) (18,88)
        Polygon (11,97) (17,93) (21,101) (24,100)
        Ellipse (39,43 3x5)
        Ellipse (55,43 1x5)
        Line (45,30) (38,33)
        Line (52,31) (55,33)
        Polygon (43,54) (44,58) (53,56) (49,55)
        RoundedRectangle (41,64 10x19)
        Polygon (29,27) (58,22) (60,12) (58,9) (54,0) (45,2) (39,3) (35,9) (36,16) (45,14) (48,9) (46,6) (42,12)
        Polygon (25,28) (9,48) (11,53) (15,56) (19,57) (26,56) (28,50) (32,43) (27,42) (22,43) (17,48) (17,48) (22,49)
        Polygon (34,12) (6,9) (0,47) (4,50) (8,51) (15,50) (17,44) (21,37) (16,36) (11,37) (6,42) (6,42) (11,43)
        Polygon (36,63) (28,68) (31,80) (47,72)
    Group (170,218 61x89)
        Ellipse (0,0 58x79)
        Line (39,85) (37,76)
        Polygon (36,87) (42,83) (48,86) (48,84)
        Polygon (50,68) (48,67) (61,65) (55,55)
        Line (13,84) (16,76)
        Polygon (9,85) (15,81) (19,89) (22,88)
        Ellipse (37,31 3x5)
        Ellipse (53,31 1x5)
        Line (41,20) (36,21)
        Line (50,19) (53,21)
        RoundedRectangle (35,30 11x9)
        Polygon (26,53) (22,56) (22,68) (24,70)
        RoundedRectangle (50,30 8x8)
        Line (50,34) (46,34)
    Group (174,538 74x85)
        Line (42,81) (40,72)
        Polygon (39,83) (45,79) (51,82) (51,80)
        Ellipse (0,0 58x79)
        Polygon (56,62) (51,55) (74,54) (58,43)
        Polygon (24,47) (21,53) (20,66) (22,62)
        Line (16,80) (19,72)
        Polygon (12,81) (18,77) (22,85) (25,84)
        Polygon (44,39) (54,48) (56,37) (57,39)
        Ellipse (39,26 4x6)
        Ellipse (55,26 2x6)
        Line (43,15) (36,17)
        Line (50,15) (55,17)
    Group (168,1791 75x89)
        Line (43,85) (41,76)
        Polygon (40,87) (46,83) (52,86) (52,84)
        Ellipse (2,0 58x79)
        Polygon (53,65) (52,59) (75,58) (59,47)
        Polygon (24,52) (25,58) (27,67) (33,45)
        Line (17,84) (20,76)
        Polygon (13,85) (19,81) (23,89) (26,88)
        Rectangle (0,11 26x31)
        Rectangle (0,0 54x15)
        Ellipse (40,30 4x6)
        Ellipse (56,30 2x6)
        Line (44,21) (37,21)
        Line (50,20) (58,21)
        Rectangle (44,41 12x4)
    Rectangle (1924,-301 135x76)
    Rectangle (17,1814 86x72), "B1 F"
    Rectangle (4,1509 86x72), "1 F"
    Rectangle (8,1183 86x72), "2 F"
    Rectangle (10,878 86x72), "3 F"
    Rectangle (8,560 86x72), "4 F"
    Rectangle (6,241 86x72), "5 F"
    Frame (9,1277 319x161)
        shows OutsideEle(fbFloorsVisu := PLC_PRG.fbFloors[1])
    Frame (8,956 319x161)
        shows OutsideEle(fbFloorsVisu := PLC_PRG.fbFloors[2])
    Frame (16,1589 319x161)
        shows OutsideEle(fbFloorsVisu := PLC_PRG.fbFloors[0])
    Frame (9,636 319x161)
        shows OutsideEle(fbFloorsVisu := PLC_PRG.fbFloors[3])
    Frame (5,325 319x161)
        shows OutsideEle(fbFloorsVisu := PLC_PRG.fbFloors[4])
    Frame (7,11 319x161)
        shows OutsideEle(fbFloorsVisu := PLC_PRG.fbFloors[5])
    Rectangle (5,27 66x71)
    Rectangle (15,1688 66x71)
    Frame (388,945 316x317)
        shows Elavator(fbElevatorVisu := PLC_PRG.fbElevator[1])
        p2738717112: PLC_PRG.fbElevator[1].iMove
    Frame (1588,1258 319x314)
        shows FreightElavator(fbFreightVisu := PLC_PRG.fbElevator[4])
        p2738717112: PLC_PRG.fbElevator[4].iMove
END_VISUALIZATION
